INTERFACE I_Mc3SlaveAxis EXTENDS I_Mc3Axis_PTP, I_Mc3AxisGear

END_INTERFACE

(* stored: Version 1.1.0.1, ProductVersion 3.1.4026.20
   Itf I_Mc3SlaveAxis: Id {2ca40060-2e90-4534-bf74-e0726c3baae4} *)
